// TIA Portal V20 export
TYPE "Struct_ANY"
   STRUCT
      S7 : Byte;   // 0x10
      DataType : Byte;
      Repetition : Word;
      DBNumber : Word;
      Address : DWord;   // Memory area + address
   END_STRUCT;
END_TYPE
